FUNCTION_BLOCK NodePack_PlcBasicDisplay IMPLEMENTS I_NodePack
VAR
	node_Display_BOOL : Node_Display_BOOL;
END_VAR

METHOD PUBLIC RegisterWithGraph
VAR_INPUT
	TcGraph : I_GraphFactory;
END_VAR
TcGraph.RegisterNodeByType('PLC Basic/Display/BOOL',node_Display_BOOL);
END_METHOD

END_FUNCTION_BLOCK

(* stored: Version 1.1.0.1, ProductVersion 3.1.4024.12
   POU NodePack_PlcBasicDisplay: Id {f8c90f2a-938e-0576-2379-b6509a0f06b0}, SpecialFunc None
   Method RegisterWithGraph: Id {41c9db0a-1f24-0d2a-0d64-b28dad2a40b1} *)
